// TIA Portal V17 export
// export: Created 2025-03-10T12:18:24.9535998Z, ExportSetting WithDefaults, DisplayName Totally Integrated Automation Portal, DisplayVersion V17 Update 8, DisplayName TIA Portal Openness, DisplayVersion V17 Update 8, DisplayName TIA Portal Version Control Interface, DisplayVersion V17, DisplayName SINAMICS Startdrive Advanced, DisplayVersion V17 SP2, DisplayName SINAMICS Startdrive G110M, G120, G120C, G120D, G120P, G115D, DisplayVersion V17 SP2, DisplayName SINAMICS Startdrive G130, G150, S120, S150, SINAMICS MV, S210, DisplayVersion V17 SP2, DisplayName STEP 7 Professional, DisplayVersion V17 Update 8, DisplayName SINUMERIK ONE STEP 7 Toolbox, DisplayVersion V17 Update 12, DisplayName SINUMERIK 840D sl STEP 7 Toolbox, DisplayVersion V17 Update 12, DisplayName STEP 7 Safety, DisplayVersion V17 Update 6, DisplayName WinCC Advanced, DisplayVersion V17 Update 8
DATA_BLOCK "DB428_OPERATOR_HELP"   // DB428
{ S7_Optimized_Access := 'FALSE' }
VERSION : 1.0
// stored: AutoNumber false, DBAccessibleFromOPCUA true, DBAccessibleFromWebserver true, IsOnlyStoredInLoadMemory false, IsWriteProtectedInAS false
   VAR RETAIN
      HELP_OPERATOR_0 : Bool;   // EMPTY
      HELP_OPERATOR_1 : Bool;   // EMPTY
      HELP_OPERATOR_2 : Bool;
      HELP_OPERATOR_3 : Bool;
      HELP_OPERATOR_4 : Bool;
      HELP_OPERATOR_5 : Bool;
      HELP_OPERATOR_6 : Bool;
      HELP_OPERATOR_7 : Bool;
      HELP_OPERATOR_8 : Bool;
      HELP_OPERATOR_9 : Bool;
      HELP_OPERATOR_10 : Bool;
      HELP_OPERATOR_11 : Bool;
      HELP_OPERATOR_12 : Bool;
      HELP_OPERATOR_13 : Bool;
      HELP_OPERATOR_14 : Bool;
      HELP_OPERATOR_15 : Bool;
      HELP_OPERATOR_16 : Bool;
      HELP_OPERATOR_17 : Bool;
      HELP_OPERATOR_18 : Bool;
      HELP_OPERATOR_19 : Bool;
      HELP_OPERATOR_20 : Bool;
      HELP_OPERATOR_21 : Bool;
      HELP_OPERATOR_22 : Bool;
      HELP_OPERATOR_23 : Bool;
      HELP_OPERATOR_24 : Bool;
      HELP_OPERATOR_25 : Bool;
      HELP_OPERATOR_26 : Bool;
      HELP_OPERATOR_27 : Bool;
      HELP_OPERATOR_28 : Bool;
      HELP_OPERATOR_29 : Bool;
      HELP_OPERATOR_30 : Bool;
      HELP_OPERATOR_31 : Bool;
      HELP_OPERATOR_32 : Bool;
      HELP_OPERATOR_33 : Bool;
      HELP_OPERATOR_34 : Bool;
      HELP_OPERATOR_35 : Bool;
      HELP_OPERATOR_36 : Bool;
      HELP_OPERATOR_37 : Bool;
      HELP_OPERATOR_38 : Bool;
      HELP_OPERATOR_39 : Bool;
      HELP_OPERATOR_40 : Bool;
      HELP_OPERATOR_41 : Bool;
      HELP_OPERATOR_42 : Bool;
      HELP_OPERATOR_43 : Bool;
      HELP_OPERATOR_44 : Bool;
      HELP_OPERATOR_45 : Bool;
      HELP_OPERATOR_46 : Bool;
      HELP_OPERATOR_47 : Bool;
      HELP_OPERATOR_48 : Bool;
      HELP_OPERATOR_49 : Bool;
      HELP_OPERATOR_50 : Bool;
      HELP_OPERATOR_51 : Bool;
      HELP_OPERATOR_52 : Bool;
      HELP_OPERATOR_53 : Bool;
      HELP_OPERATOR_54 : Bool;
      HELP_OPERATOR_55 : Bool;
      HELP_OPERATOR_56 : Bool;
      HELP_OPERATOR_57 : Bool;
      HELP_OPERATOR_58 : Bool;
      HELP_OPERATOR_59 : Bool;
      HELP_OPERATOR_60 : Bool;
      HELP_OPERATOR_61 : Bool;
      HELP_OPERATOR_62 : Bool;
      HELP_OPERATOR_63 : Bool;
      HELP_OPERATOR_64 : Bool;
      HELP_OPERATOR_65 : Bool;
      HELP_OPERATOR_66 : Bool;
      HELP_OPERATOR_67 : Bool;
      HELP_OPERATOR_68 : Bool;
      HELP_OPERATOR_69 : Bool;
      HELP_OPERATOR_70 : Bool;
      HELP_OPERATOR_71 : Bool;
      HELP_OPERATOR_72 : Bool;
      HELP_OPERATOR_73 : Bool;
      HELP_OPERATOR_74 : Bool;
      HELP_OPERATOR_75 : Bool;
      HELP_OPERATOR_76 : Bool;
      HELP_OPERATOR_77 : Bool;
      HELP_OPERATOR_78 : Bool;
      HELP_OPERATOR_79 : Bool;
      HELP_OPERATOR_80 : Bool;
      HELP_OPERATOR_81 : Bool;
      HELP_OPERATOR_82 : Bool;
      HELP_OPERATOR_83 : Bool;
      HELP_OPERATOR_84 : Bool;
      HELP_OPERATOR_85 : Bool;
      HELP_OPERATOR_86 : Bool;
      HELP_OPERATOR_87 : Bool;
      HELP_OPERATOR_88 : Bool;
      HELP_OPERATOR_89 : Bool;
      HELP_OPERATOR_90 : Bool;
      HELP_OPERATOR_91 : Bool;
      HELP_OPERATOR_92 : Bool;
      HELP_OPERATOR_93 : Bool;
      HELP_OPERATOR_94 : Bool;
      HELP_OPERATOR_95 : Bool;
      HELP_OPERATOR_96 : Bool;
      HELP_OPERATOR_97 : Bool;
      HELP_OPERATOR_98 : Bool;
      HELP_OPERATOR_99 : Bool;
      HELP_OPERATOR_100 : Bool;
      HELP_OPERATOR_101 : Bool;
      HELP_OPERATOR_102 : Bool;
      HELP_OPERATOR_103 : Bool;
      HELP_OPERATOR_104 : Bool;
      HELP_OPERATOR_105 : Bool;
      HELP_OPERATOR_106 : Bool;
      HELP_OPERATOR_107 : Bool;
      HELP_OPERATOR_108 : Bool;
      HELP_OPERATOR_109 : Bool;
      HELP_OPERATOR_110 : Bool;
      HELP_OPERATOR_111 : Bool;
      HELP_OPERATOR_112 : Bool;
      HELP_OPERATOR_113 : Bool;
      HELP_OPERATOR_114 : Bool;
      HELP_OPERATOR_115 : Bool;
      HELP_OPERATOR_116 : Bool;
      HELP_OPERATOR_117 : Bool;
      HELP_OPERATOR_118 : Bool;
      HELP_OPERATOR_119 : Bool;
      HELP_OPERATOR_120 : Bool;
      HELP_OPERATOR_121 : Bool;
      HELP_OPERATOR_122 : Bool;
      HELP_OPERATOR_123 : Bool;
      HELP_OPERATOR_124 : Bool;
      HELP_OPERATOR_125 : Bool;
      HELP_OPERATOR_126 : Bool;
      HELP_OPERATOR_127 : Bool;
      HELP_OPERATOR_128 : Bool;
      HELP_OPERATOR_129 : Bool;
      HELP_OPERATOR_130 : Bool;
      HELP_OPERATOR_131 : Bool;
      HELP_OPERATOR_132 : Bool;
      HELP_OPERATOR_133 : Bool;
      HELP_OPERATOR_134 : Bool;
      HELP_OPERATOR_135 : Bool;
      HELP_OPERATOR_136 : Bool;
      HELP_OPERATOR_137 : Bool;
      HELP_OPERATOR_138 : Bool;
      HELP_OPERATOR_139 : Bool;
      HELP_OPERATOR_140 : Bool;
      HELP_OPERATOR_141 : Bool;
      HELP_OPERATOR_142 : Bool;
      HELP_OPERATOR_143 : Bool;
      HELP_OPERATOR_144 : Bool;
      HELP_OPERATOR_145 : Bool;
      HELP_OPERATOR_146 : Bool;
      HELP_OPERATOR_147 : Bool;
      HELP_OPERATOR_148 : Bool;
      HELP_OPERATOR_149 : Bool;
      HELP_OPERATOR_150 : Bool;   // RETURN UNIT 1 TO HOME POSITION
      HELP_OPERATOR_151 : Bool;   // RETURN UNIT 2 TO HOME POSITION
      HELP_OPERATOR_152 : Bool;   // RETURN UNIT 3 TO HOME POSITION
      HELP_OPERATOR_153 : Bool;   // RETURN UNIT 4 TO HOME POSITION
      HELP_OPERATOR_154 : Bool;   // RETURN UNIT 5 TO HOME POSITION
      HELP_OPERATOR_155 : Bool;   // RETURN UNIT 6 TO HOME POSITION
      HELP_OPERATOR_156 : Bool;   // RETURN UNIT 7 TO HOME POSITION
      HELP_OPERATOR_157 : Bool;   // RETURN UNIT 8 TO HOME POSITION
      HELP_OPERATOR_158 : Bool;   // RETURN UNIT 9 TO HOME POSITION
      HELP_OPERATOR_159 : Bool;   // RETURN UNIT 10 TO HOME POSITION
      HELP_OPERATOR_160 : Bool;
      HELP_OPERATOR_161 : Bool;
      HELP_OPERATOR_162 : Bool;   // UNIT 1 IN HOME POSITION
      HELP_OPERATOR_163 : Bool;   // UNIT 2 IN HOME POSITION
      HELP_OPERATOR_164 : Bool;   // UNIT 3 IN HOME POSITION
      HELP_OPERATOR_165 : Bool;   // UNIT 4 IN HOME POSITION
      HELP_OPERATOR_166 : Bool;   // UNIT 5 IN HOME POSITION
      HELP_OPERATOR_167 : Bool;   // UNIT 6 IN HOME POSITION
      HELP_OPERATOR_168 : Bool;   // UNIT 7 IN HOME POSITION
      HELP_OPERATOR_169 : Bool;   // UNIT 8 IN HOME POSITION
      HELP_OPERATOR_170 : Bool;   // UNIT 9 IN HOME POSITION
      HELP_OPERATOR_171 : Bool;   // UNIT 10 IN HOME POSITION
      HELP_OPERATOR_172 : Bool;
      HELP_OPERATOR_173 : Bool;
      HELP_OPERATOR_174 : Bool;   // UNIT 01R SPINDLES NOT STOPPED
      HELP_OPERATOR_175 : Bool;   // UNIT 01L SPINDLES NOT STOPPED
      HELP_OPERATOR_176 : Bool;
      HELP_OPERATOR_177 : Bool;
      HELP_OPERATOR_178 : Bool;   // TOOLS IN MAGAZINE 01R NOT OK
      HELP_OPERATOR_179 : Bool;   // TOOLS IN MAGAZINE 01L NOT OK
      HELP_OPERATOR_180 : Bool;
      HELP_OPERATOR_181 : Bool;
      HELP_OPERATOR_182 : Bool;   // RETURN MACHINE TO HOME POSITION
      HELP_OPERATOR_183 : Bool;
      HELP_OPERATOR_184 : Bool;   // RETURN PART HANDLING DEVICE TO HOME POSITION
      HELP_OPERATOR_185 : Bool;   // PART HANDLING DEVICE IN HOME POSITION
      HELP_OPERATOR_186 : Bool;   // ADVANCE PHD TO LOAD UNLOAD POS FIXTURE
      HELP_OPERATOR_187 : Bool;
      HELP_OPERATOR_188 : Bool;
      HELP_OPERATOR_189 : Bool;
      HELP_OPERATOR_190 : Bool;   // NO PART AT FEED
      HELP_OPERATOR_191 : Bool;   // PARTS DELIVERY OCCUPIED
      HELP_OPERATOR_192 : Bool;
      HELP_OPERATOR_193 : Bool;
      HELP_OPERATOR_194 : Bool;
      HELP_OPERATOR_195 : Bool;
      HELP_OPERATOR_196 : Bool;
      HELP_OPERATOR_197 : Bool;
      HELP_OPERATOR_198 : Bool;
      HELP_OPERATOR_199 : Bool;
      HELP_OPERATOR_200 : Bool;   // SELECT MANUAL MODE
      HELP_OPERATOR_201 : Bool;   // SELECT JOG MODE
      HELP_OPERATOR_202 : Bool;   // SELECT SEMIAUTOMATIC MODE
      HELP_OPERATOR_203 : Bool;   // SELECT TOOL CHANGE MODE
      HELP_OPERATOR_204 : Bool;   // SELECT AUTOMATIC MODE
      HELP_OPERATOR_205 : Bool;   // SELECT INCREMENTAL MODE
      HELP_OPERATOR_206 : Bool;   // SELECT AUTO. OR SEMIAUTO. OR SINGLE MODE
      HELP_OPERATOR_207 : Bool;
      HELP_OPERATOR_208 : Bool;
      HELP_OPERATOR_209 : Bool;
      HELP_OPERATOR_210 : Bool;
      HELP_OPERATOR_211 : Bool;
      HELP_OPERATOR_212 : Bool;
      HELP_OPERATOR_213 : Bool;
      HELP_OPERATOR_214 : Bool;
      HELP_OPERATOR_215 : Bool;   // UNSELECT REFERENCE MODE
      HELP_OPERATOR_216 : Bool;   // UNSELECT STEP BY STEP MODE
      HELP_OPERATOR_217 : Bool;   // UNSELECT MANUAL LOADING CYCLE
      HELP_OPERATOR_218 : Bool;   // UNSELECT MDA MODE
      HELP_OPERATOR_219 : Bool;   // UNSELECT RUN-OUT CYCLE
      HELP_OPERATOR_220 : Bool;   // UNSELECT DRY CYCLE
      HELP_OPERATOR_221 : Bool;   // UNSELECT GANTRY TEST CYCLE
      HELP_OPERATOR_222 : Bool;   // UNSELECT ROBOT DRY CYCLE
      HELP_OPERATOR_223 : Bool;   // UNSELECT SINGLE CYCLE
      HELP_OPERATOR_224 : Bool;
      HELP_OPERATOR_225 : Bool;
      HELP_OPERATOR_226 : Bool;
      HELP_OPERATOR_227 : Bool;
      HELP_OPERATOR_228 : Bool;
      HELP_OPERATOR_229 : Bool;
      HELP_OPERATOR_230 : Bool;   // ENABLE BA1 MODE
      HELP_OPERATOR_231 : Bool;   // ENABLE BA1 OR BA3 MODE
      HELP_OPERATOR_232 : Bool;   // ENABLE BA2 MODE OR CLOSE SAFETY DOORS
      HELP_OPERATOR_233 : Bool;
      HELP_OPERATOR_234 : Bool;
      HELP_OPERATOR_235 : Bool;
      HELP_OPERATOR_236 : Bool;
      HELP_OPERATOR_237 : Bool;
      HELP_OPERATOR_238 : Bool;
      HELP_OPERATOR_239 : Bool;
      HELP_OPERATOR_240 : Bool;
      HELP_OPERATOR_241 : Bool;
      HELP_OPERATOR_242 : Bool;
      HELP_OPERATOR_243 : Bool;
      HELP_OPERATOR_244 : Bool;
      HELP_OPERATOR_245 : Bool;
      HELP_OPERATOR_246 : Bool;
      HELP_OPERATOR_247 : Bool;
      HELP_OPERATOR_248 : Bool;
      HELP_OPERATOR_249 : Bool;
      HELP_OPERATOR_250 : Bool;   // MAIN OPERATOR PANEL, PRESS BUTTON CONTROL ON
      HELP_OPERATOR_251 : Bool;   // MAIN OPERATOR PANEL, PRESS BUTTON RESET
      HELP_OPERATOR_252 : Bool;   // REMOVE EMERGENCY STOPS, PRESS RESET FAULTS
      HELP_OPERATOR_253 : Bool;   // MACHINE STOP SERVICES DELAYED ENABLED
      HELP_OPERATOR_254 : Bool;   // SWITCH ON PNEUMATIC SYSTEM
      HELP_OPERATOR_255 : Bool;
      HELP_OPERATOR_256 : Bool;
      HELP_OPERATOR_257 : Bool;
      HELP_OPERATOR_258 : Bool;
      HELP_OPERATOR_259 : Bool;
      HELP_OPERATOR_260 : Bool;
      HELP_OPERATOR_261 : Bool;
      HELP_OPERATOR_262 : Bool;
      HELP_OPERATOR_263 : Bool;
      HELP_OPERATOR_264 : Bool;
      HELP_OPERATOR_265 : Bool;
      HELP_OPERATOR_266 : Bool;
      HELP_OPERATOR_267 : Bool;
      HELP_OPERATOR_268 : Bool;
      HELP_OPERATOR_269 : Bool;
      HELP_OPERATOR_270 : Bool;
      HELP_OPERATOR_271 : Bool;
      HELP_OPERATOR_272 : Bool;
      HELP_OPERATOR_273 : Bool;
      HELP_OPERATOR_274 : Bool;
      HELP_OPERATOR_275 : Bool;
      HELP_OPERATOR_276 : Bool;
      HELP_OPERATOR_277 : Bool;
      HELP_OPERATOR_278 : Bool;
      HELP_OPERATOR_279 : Bool;
      HELP_OPERATOR_280 : Bool;
      HELP_OPERATOR_281 : Bool;
      HELP_OPERATOR_282 : Bool;
      HELP_OPERATOR_283 : Bool;
      HELP_OPERATOR_284 : Bool;
      HELP_OPERATOR_285 : Bool;
      HELP_OPERATOR_286 : Bool;
      HELP_OPERATOR_287 : Bool;
      HELP_OPERATOR_288 : Bool;
      HELP_OPERATOR_289 : Bool;
      HELP_OPERATOR_290 : Bool;
      HELP_OPERATOR_291 : Bool;
      HELP_OPERATOR_292 : Bool;
      HELP_OPERATOR_293 : Bool;
      HELP_OPERATOR_294 : Bool;
      HELP_OPERATOR_295 : Bool;
      HELP_OPERATOR_296 : Bool;
      HELP_OPERATOR_297 : Bool;
      HELP_OPERATOR_298 : Bool;
      HELP_OPERATOR_299 : Bool;
      HELP_OPERATOR_300 : Bool;
      HELP_OPERATOR_301 : Bool;
      HELP_OPERATOR_302 : Bool;
      HELP_OPERATOR_303 : Bool;
      HELP_OPERATOR_304 : Bool;
      HELP_OPERATOR_305 : Bool;
      HELP_OPERATOR_306 : Bool;
      HELP_OPERATOR_307 : Bool;
      HELP_OPERATOR_308 : Bool;
      HELP_OPERATOR_309 : Bool;
      HELP_OPERATOR_310 : Bool;
      HELP_OPERATOR_311 : Bool;
      HELP_OPERATOR_312 : Bool;
      HELP_OPERATOR_313 : Bool;
      HELP_OPERATOR_314 : Bool;
      HELP_OPERATOR_315 : Bool;
      HELP_OPERATOR_316 : Bool;
      HELP_OPERATOR_317 : Bool;
      HELP_OPERATOR_318 : Bool;
      HELP_OPERATOR_319 : Bool;
      HELP_OPERATOR_320 : Bool;
      HELP_OPERATOR_321 : Bool;
      HELP_OPERATOR_322 : Bool;
      HELP_OPERATOR_323 : Bool;
      HELP_OPERATOR_324 : Bool;
      HELP_OPERATOR_325 : Bool;
      HELP_OPERATOR_326 : Bool;
      HELP_OPERATOR_327 : Bool;
      HELP_OPERATOR_328 : Bool;
      HELP_OPERATOR_329 : Bool;
      HELP_OPERATOR_330 : Bool;
      HELP_OPERATOR_331 : Bool;
      HELP_OPERATOR_332 : Bool;
      HELP_OPERATOR_333 : Bool;
      HELP_OPERATOR_334 : Bool;
      HELP_OPERATOR_335 : Bool;
      HELP_OPERATOR_336 : Bool;
      HELP_OPERATOR_337 : Bool;
      HELP_OPERATOR_338 : Bool;
      HELP_OPERATOR_339 : Bool;
      HELP_OPERATOR_340 : Bool;
      HELP_OPERATOR_341 : Bool;
      HELP_OPERATOR_342 : Bool;
      HELP_OPERATOR_343 : Bool;
      HELP_OPERATOR_344 : Bool;
      HELP_OPERATOR_345 : Bool;
      HELP_OPERATOR_346 : Bool;
      HELP_OPERATOR_347 : Bool;
      HELP_OPERATOR_348 : Bool;
      HELP_OPERATOR_349 : Bool;
      HELP_OPERATOR_350 : Bool;
      HELP_OPERATOR_351 : Bool;
      HELP_OPERATOR_352 : Bool;
      HELP_OPERATOR_353 : Bool;
      HELP_OPERATOR_354 : Bool;
      HELP_OPERATOR_355 : Bool;
      HELP_OPERATOR_356 : Bool;
      HELP_OPERATOR_357 : Bool;
      HELP_OPERATOR_358 : Bool;
      HELP_OPERATOR_359 : Bool;
      HELP_OPERATOR_360 : Bool;
      HELP_OPERATOR_361 : Bool;
      HELP_OPERATOR_362 : Bool;
      HELP_OPERATOR_363 : Bool;
      HELP_OPERATOR_364 : Bool;
      HELP_OPERATOR_365 : Bool;
      HELP_OPERATOR_366 : Bool;
      HELP_OPERATOR_367 : Bool;
      HELP_OPERATOR_368 : Bool;
      HELP_OPERATOR_369 : Bool;
      HELP_OPERATOR_370 : Bool;
      HELP_OPERATOR_371 : Bool;
      HELP_OPERATOR_372 : Bool;
      HELP_OPERATOR_373 : Bool;
      HELP_OPERATOR_374 : Bool;
      HELP_OPERATOR_375 : Bool;
      HELP_OPERATOR_376 : Bool;
      HELP_OPERATOR_377 : Bool;
      HELP_OPERATOR_378 : Bool;
      HELP_OPERATOR_379 : Bool;
      HELP_OPERATOR_380 : Bool;
      HELP_OPERATOR_381 : Bool;
      HELP_OPERATOR_382 : Bool;
      HELP_OPERATOR_383 : Bool;
      HELP_OPERATOR_384 : Bool;
      HELP_OPERATOR_385 : Bool;
      HELP_OPERATOR_386 : Bool;
      HELP_OPERATOR_387 : Bool;
      HELP_OPERATOR_388 : Bool;
      HELP_OPERATOR_389 : Bool;
      HELP_OPERATOR_390 : Bool;
      HELP_OPERATOR_391 : Bool;
      HELP_OPERATOR_392 : Bool;
      HELP_OPERATOR_393 : Bool;
      HELP_OPERATOR_394 : Bool;
      HELP_OPERATOR_395 : Bool;
      HELP_OPERATOR_396 : Bool;
      HELP_OPERATOR_397 : Bool;
      HELP_OPERATOR_398 : Bool;
      HELP_OPERATOR_399 : Bool;
      HELP_OPERATOR_400 : Bool;
      HELP_OPERATOR_401 : Bool;
      HELP_OPERATOR_402 : Bool;
      HELP_OPERATOR_403 : Bool;
      HELP_OPERATOR_404 : Bool;
      HELP_OPERATOR_405 : Bool;
      HELP_OPERATOR_406 : Bool;
      HELP_OPERATOR_407 : Bool;
      HELP_OPERATOR_408 : Bool;
      HELP_OPERATOR_409 : Bool;
      HELP_OPERATOR_410 : Bool;
      HELP_OPERATOR_411 : Bool;
      HELP_OPERATOR_412 : Bool;
      HELP_OPERATOR_413 : Bool;
      HELP_OPERATOR_414 : Bool;
      HELP_OPERATOR_415 : Bool;
      HELP_OPERATOR_416 : Bool;
      HELP_OPERATOR_417 : Bool;
      HELP_OPERATOR_418 : Bool;
      HELP_OPERATOR_419 : Bool;
      HELP_OPERATOR_420 : Bool;
      HELP_OPERATOR_421 : Bool;
      HELP_OPERATOR_422 : Bool;
      HELP_OPERATOR_423 : Bool;
      HELP_OPERATOR_424 : Bool;
      HELP_OPERATOR_425 : Bool;
      HELP_OPERATOR_426 : Bool;
      HELP_OPERATOR_427 : Bool;
      HELP_OPERATOR_428 : Bool;
      HELP_OPERATOR_429 : Bool;
      HELP_OPERATOR_430 : Bool;
      HELP_OPERATOR_431 : Bool;
      HELP_OPERATOR_432 : Bool;
      HELP_OPERATOR_433 : Bool;
      HELP_OPERATOR_434 : Bool;
      HELP_OPERATOR_435 : Bool;
      HELP_OPERATOR_436 : Bool;
      HELP_OPERATOR_437 : Bool;
      HELP_OPERATOR_438 : Bool;
      HELP_OPERATOR_439 : Bool;
      HELP_OPERATOR_440 : Bool;
      HELP_OPERATOR_441 : Bool;
      HELP_OPERATOR_442 : Bool;
      HELP_OPERATOR_443 : Bool;
      HELP_OPERATOR_444 : Bool;
      HELP_OPERATOR_445 : Bool;
      HELP_OPERATOR_446 : Bool;
      HELP_OPERATOR_447 : Bool;
      HELP_OPERATOR_448 : Bool;
      HELP_OPERATOR_449 : Bool;
      HELP_OPERATOR_450 : Bool;
      HELP_OPERATOR_451 : Bool;
      HELP_OPERATOR_452 : Bool;
      HELP_OPERATOR_453 : Bool;
      HELP_OPERATOR_454 : Bool;
      HELP_OPERATOR_455 : Bool;
      HELP_OPERATOR_456 : Bool;
      HELP_OPERATOR_457 : Bool;
      HELP_OPERATOR_458 : Bool;
      HELP_OPERATOR_459 : Bool;
      HELP_OPERATOR_460 : Bool;
      HELP_OPERATOR_461 : Bool;
      HELP_OPERATOR_462 : Bool;
      HELP_OPERATOR_463 : Bool;
      HELP_OPERATOR_464 : Bool;
      HELP_OPERATOR_465 : Bool;
      HELP_OPERATOR_466 : Bool;
      HELP_OPERATOR_467 : Bool;
      HELP_OPERATOR_468 : Bool;
      HELP_OPERATOR_469 : Bool;
      HELP_OPERATOR_470 : Bool;
      HELP_OPERATOR_471 : Bool;
      HELP_OPERATOR_472 : Bool;
      HELP_OPERATOR_473 : Bool;
      HELP_OPERATOR_474 : Bool;
      HELP_OPERATOR_475 : Bool;
      HELP_OPERATOR_476 : Bool;
      HELP_OPERATOR_477 : Bool;
      HELP_OPERATOR_478 : Bool;
      HELP_OPERATOR_479 : Bool;
      HELP_OPERATOR_480 : Bool;
      HELP_OPERATOR_481 : Bool;
      HELP_OPERATOR_482 : Bool;
      HELP_OPERATOR_483 : Bool;
      HELP_OPERATOR_484 : Bool;
      HELP_OPERATOR_485 : Bool;
      HELP_OPERATOR_486 : Bool;
      HELP_OPERATOR_487 : Bool;
      HELP_OPERATOR_488 : Bool;
      HELP_OPERATOR_489 : Bool;
      HELP_OPERATOR_490 : Bool;
      HELP_OPERATOR_491 : Bool;
      HELP_OPERATOR_492 : Bool;
      HELP_OPERATOR_493 : Bool;
      HELP_OPERATOR_494 : Bool;
      HELP_OPERATOR_495 : Bool;
      HELP_OPERATOR_496 : Bool;
      HELP_OPERATOR_497 : Bool;
      HELP_OPERATOR_498 : Bool;
      HELP_OPERATOR_499 : Bool;
      HELP_OPERATOR_500 : Bool;
      HELP_OPERATOR_501 : Bool;
      HELP_OPERATOR_502 : Bool;
      HELP_OPERATOR_503 : Bool;
      HELP_OPERATOR_504 : Bool;
      HELP_OPERATOR_505 : Bool;
      HELP_OPERATOR_506 : Bool;
      HELP_OPERATOR_507 : Bool;
      HELP_OPERATOR_508 : Bool;
      HELP_OPERATOR_509 : Bool;
      HELP_OPERATOR_510 : Bool;
      HELP_OPERATOR_511 : Bool;
      HELP_OPERATOR_512 : Bool;
      HELP_OPERATOR_513 : Bool;
      HELP_OPERATOR_514 : Bool;
      HELP_OPERATOR_515 : Bool;
      HELP_OPERATOR_516 : Bool;
      HELP_OPERATOR_517 : Bool;
      HELP_OPERATOR_518 : Bool;
      HELP_OPERATOR_519 : Bool;
      HELP_OPERATOR_520 : Bool;
      HELP_OPERATOR_521 : Bool;
      HELP_OPERATOR_522 : Bool;
      HELP_OPERATOR_523 : Bool;
      HELP_OPERATOR_524 : Bool;
      HELP_OPERATOR_525 : Bool;
      HELP_OPERATOR_526 : Bool;
      HELP_OPERATOR_527 : Bool;
      HELP_OPERATOR_528 : Bool;
      HELP_OPERATOR_529 : Bool;
      HELP_OPERATOR_530 : Bool;
      HELP_OPERATOR_531 : Bool;   // STIRRER MOTOR NOT ENABLED
      HELP_OPERATOR_532 : Bool;   // STIRRER FAULT
      HELP_OPERATOR_533 : Bool;   // STIRRER ON
      HELP_OPERATOR_534 : Bool;   // STIRRER STOP GENERAL CONDITIONS MISSING
      HELP_OPERATOR_535 : Bool;   // STIRRER OFF
      HELP_OPERATOR_536 : Bool;
      HELP_OPERATOR_537 : Bool;
      HELP_OPERATOR_538 : Bool;
      HELP_OPERATOR_539 : Bool;
      HELP_OPERATOR_540 : Bool;   // TEMPERATURE JACKET BREAKER TRIPPED
      HELP_OPERATOR_541 : Bool;
      HELP_OPERATOR_542 : Bool;
      HELP_OPERATOR_543 : Bool;
      HELP_OPERATOR_544 : Bool;
      HELP_OPERATOR_545 : Bool;
      HELP_OPERATOR_546 : Bool;
      HELP_OPERATOR_547 : Bool;
      HELP_OPERATOR_548 : Bool;
      HELP_OPERATOR_549 : Bool;
      HELP_OPERATOR_550 : Bool;
      HELP_OPERATOR_551 : Bool;
      HELP_OPERATOR_552 : Bool;
      HELP_OPERATOR_553 : Bool;
      HELP_OPERATOR_554 : Bool;
      HELP_OPERATOR_555 : Bool;
      HELP_OPERATOR_556 : Bool;
      HELP_OPERATOR_557 : Bool;
      HELP_OPERATOR_558 : Bool;
      HELP_OPERATOR_559 : Bool;
      HELP_OPERATOR_560 : Bool;
      HELP_OPERATOR_561 : Bool;
      HELP_OPERATOR_562 : Bool;
      HELP_OPERATOR_563 : Bool;
      HELP_OPERATOR_564 : Bool;
      HELP_OPERATOR_565 : Bool;
      HELP_OPERATOR_566 : Bool;
      HELP_OPERATOR_567 : Bool;
      HELP_OPERATOR_568 : Bool;
      HELP_OPERATOR_569 : Bool;
      HELP_OPERATOR_570 : Bool;
      HELP_OPERATOR_571 : Bool;
      HELP_OPERATOR_572 : Bool;
      HELP_OPERATOR_573 : Bool;
      HELP_OPERATOR_574 : Bool;
      HELP_OPERATOR_575 : Bool;
      HELP_OPERATOR_576 : Bool;
      HELP_OPERATOR_577 : Bool;
      HELP_OPERATOR_578 : Bool;
      HELP_OPERATOR_579 : Bool;
      HELP_OPERATOR_580 : Bool;
      HELP_OPERATOR_581 : Bool;
      HELP_OPERATOR_582 : Bool;
      HELP_OPERATOR_583 : Bool;
      HELP_OPERATOR_584 : Bool;
      HELP_OPERATOR_585 : Bool;
      HELP_OPERATOR_586 : Bool;
      HELP_OPERATOR_587 : Bool;
      HELP_OPERATOR_588 : Bool;
      HELP_OPERATOR_589 : Bool;
      HELP_OPERATOR_590 : Bool;
      HELP_OPERATOR_591 : Bool;
      HELP_OPERATOR_592 : Bool;
      HELP_OPERATOR_593 : Bool;
      HELP_OPERATOR_594 : Bool;
      HELP_OPERATOR_595 : Bool;
      HELP_OPERATOR_596 : Bool;
      HELP_OPERATOR_597 : Bool;
      HELP_OPERATOR_598 : Bool;
      HELP_OPERATOR_599 : Bool;
      HELP_OPERATOR_600 : Bool;
      HELP_OPERATOR_601 : Bool;
      HELP_OPERATOR_602 : Bool;
      HELP_OPERATOR_603 : Bool;
      HELP_OPERATOR_604 : Bool;
      HELP_OPERATOR_605 : Bool;
      HELP_OPERATOR_606 : Bool;
      HELP_OPERATOR_607 : Bool;
      HELP_OPERATOR_608 : Bool;
      HELP_OPERATOR_609 : Bool;
      HELP_OPERATOR_610 : Bool;
      HELP_OPERATOR_611 : Bool;
      HELP_OPERATOR_612 : Bool;
      HELP_OPERATOR_613 : Bool;
      HELP_OPERATOR_614 : Bool;
      HELP_OPERATOR_615 : Bool;
      HELP_OPERATOR_616 : Bool;
      HELP_OPERATOR_617 : Bool;
      HELP_OPERATOR_618 : Bool;
      HELP_OPERATOR_619 : Bool;
      HELP_OPERATOR_620 : Bool;
      HELP_OPERATOR_621 : Bool;
      HELP_OPERATOR_622 : Bool;
      HELP_OPERATOR_623 : Bool;
      HELP_OPERATOR_624 : Bool;
      HELP_OPERATOR_625 : Bool;
      HELP_OPERATOR_626 : Bool;
      HELP_OPERATOR_627 : Bool;
      HELP_OPERATOR_628 : Bool;
      HELP_OPERATOR_629 : Bool;
      HELP_OPERATOR_630 : Bool;
      HELP_OPERATOR_631 : Bool;
      HELP_OPERATOR_632 : Bool;
      HELP_OPERATOR_633 : Bool;
      HELP_OPERATOR_634 : Bool;
      HELP_OPERATOR_635 : Bool;
      HELP_OPERATOR_636 : Bool;
      HELP_OPERATOR_637 : Bool;
      HELP_OPERATOR_638 : Bool;
      HELP_OPERATOR_639 : Bool;
      HELP_OPERATOR_640 : Bool;
      HELP_OPERATOR_641 : Bool;
      HELP_OPERATOR_642 : Bool;
      HELP_OPERATOR_643 : Bool;
      HELP_OPERATOR_644 : Bool;
      HELP_OPERATOR_645 : Bool;
      HELP_OPERATOR_646 : Bool;
      HELP_OPERATOR_647 : Bool;
      HELP_OPERATOR_648 : Bool;
      HELP_OPERATOR_649 : Bool;
      HELP_OPERATOR_650 : Bool;
      HELP_OPERATOR_651 : Bool;
      HELP_OPERATOR_652 : Bool;
      HELP_OPERATOR_653 : Bool;
      HELP_OPERATOR_654 : Bool;
      HELP_OPERATOR_655 : Bool;
      HELP_OPERATOR_656 : Bool;
      HELP_OPERATOR_657 : Bool;
      HELP_OPERATOR_658 : Bool;
      HELP_OPERATOR_659 : Bool;
      HELP_OPERATOR_660 : Bool;
      HELP_OPERATOR_661 : Bool;
      HELP_OPERATOR_662 : Bool;
      HELP_OPERATOR_663 : Bool;
      HELP_OPERATOR_664 : Bool;
      HELP_OPERATOR_665 : Bool;
      HELP_OPERATOR_666 : Bool;
      HELP_OPERATOR_667 : Bool;
      HELP_OPERATOR_668 : Bool;
      HELP_OPERATOR_669 : Bool;
      HELP_OPERATOR_670 : Bool;
      HELP_OPERATOR_671 : Bool;
      HELP_OPERATOR_672 : Bool;
      HELP_OPERATOR_673 : Bool;
      HELP_OPERATOR_674 : Bool;
      HELP_OPERATOR_675 : Bool;
      HELP_OPERATOR_676 : Bool;
      HELP_OPERATOR_677 : Bool;
      HELP_OPERATOR_678 : Bool;
      HELP_OPERATOR_679 : Bool;
      HELP_OPERATOR_680 : Bool;
      HELP_OPERATOR_681 : Bool;
      HELP_OPERATOR_682 : Bool;
      HELP_OPERATOR_683 : Bool;
      HELP_OPERATOR_684 : Bool;
      HELP_OPERATOR_685 : Bool;
      HELP_OPERATOR_686 : Bool;
      HELP_OPERATOR_687 : Bool;
      HELP_OPERATOR_688 : Bool;
      HELP_OPERATOR_689 : Bool;
      HELP_OPERATOR_690 : Bool;
      HELP_OPERATOR_691 : Bool;
      HELP_OPERATOR_692 : Bool;
      HELP_OPERATOR_693 : Bool;
      HELP_OPERATOR_694 : Bool;
      HELP_OPERATOR_695 : Bool;
      HELP_OPERATOR_696 : Bool;
      HELP_OPERATOR_697 : Bool;
      HELP_OPERATOR_698 : Bool;
      HELP_OPERATOR_699 : Bool;
      HELP_OPERATOR_700 : Bool;
      HELP_OPERATOR_701 : Bool;
      HELP_OPERATOR_702 : Bool;
      HELP_OPERATOR_703 : Bool;
      HELP_OPERATOR_704 : Bool;
      HELP_OPERATOR_705 : Bool;
      HELP_OPERATOR_706 : Bool;
      HELP_OPERATOR_707 : Bool;
      HELP_OPERATOR_708 : Bool;
      HELP_OPERATOR_709 : Bool;
      HELP_OPERATOR_710 : Bool;
      HELP_OPERATOR_711 : Bool;
      HELP_OPERATOR_712 : Bool;
      HELP_OPERATOR_713 : Bool;
      HELP_OPERATOR_714 : Bool;
      HELP_OPERATOR_715 : Bool;
      HELP_OPERATOR_716 : Bool;
      HELP_OPERATOR_717 : Bool;
      HELP_OPERATOR_718 : Bool;
      HELP_OPERATOR_719 : Bool;
      HELP_OPERATOR_720 : Bool;
      HELP_OPERATOR_721 : Bool;
      HELP_OPERATOR_722 : Bool;
      HELP_OPERATOR_723 : Bool;
      HELP_OPERATOR_724 : Bool;
      HELP_OPERATOR_725 : Bool;
      HELP_OPERATOR_726 : Bool;
      HELP_OPERATOR_727 : Bool;
      HELP_OPERATOR_728 : Bool;
      HELP_OPERATOR_729 : Bool;
      HELP_OPERATOR_730 : Bool;
      HELP_OPERATOR_731 : Bool;
      HELP_OPERATOR_732 : Bool;
      HELP_OPERATOR_733 : Bool;
      HELP_OPERATOR_734 : Bool;
      HELP_OPERATOR_735 : Bool;
      HELP_OPERATOR_736 : Bool;
      HELP_OPERATOR_737 : Bool;
      HELP_OPERATOR_738 : Bool;
      HELP_OPERATOR_739 : Bool;
      HELP_OPERATOR_740 : Bool;
      HELP_OPERATOR_741 : Bool;
      HELP_OPERATOR_742 : Bool;
      HELP_OPERATOR_743 : Bool;
      HELP_OPERATOR_744 : Bool;
      HELP_OPERATOR_745 : Bool;
      HELP_OPERATOR_746 : Bool;
      HELP_OPERATOR_747 : Bool;
      HELP_OPERATOR_748 : Bool;
      HELP_OPERATOR_749 : Bool;
      HELP_OPERATOR_750 : Bool;
      HELP_OPERATOR_751 : Bool;
      HELP_OPERATOR_752 : Bool;
      HELP_OPERATOR_753 : Bool;
      HELP_OPERATOR_754 : Bool;
      HELP_OPERATOR_755 : Bool;
      HELP_OPERATOR_756 : Bool;
      HELP_OPERATOR_757 : Bool;
      HELP_OPERATOR_758 : Bool;
      HELP_OPERATOR_759 : Bool;
      HELP_OPERATOR_760 : Bool;
      HELP_OPERATOR_761 : Bool;
      HELP_OPERATOR_762 : Bool;
      HELP_OPERATOR_763 : Bool;
      HELP_OPERATOR_764 : Bool;
      HELP_OPERATOR_765 : Bool;
      HELP_OPERATOR_766 : Bool;
      HELP_OPERATOR_767 : Bool;
      HELP_OPERATOR_768 : Bool;
      HELP_OPERATOR_769 : Bool;
      HELP_OPERATOR_770 : Bool;
      HELP_OPERATOR_771 : Bool;
      HELP_OPERATOR_772 : Bool;
      HELP_OPERATOR_773 : Bool;
      HELP_OPERATOR_774 : Bool;
      HELP_OPERATOR_775 : Bool;
      HELP_OPERATOR_776 : Bool;
      HELP_OPERATOR_777 : Bool;
      HELP_OPERATOR_778 : Bool;
      HELP_OPERATOR_779 : Bool;
      HELP_OPERATOR_780 : Bool;
      HELP_OPERATOR_781 : Bool;
      HELP_OPERATOR_782 : Bool;
      HELP_OPERATOR_783 : Bool;
      HELP_OPERATOR_784 : Bool;
      HELP_OPERATOR_785 : Bool;
      HELP_OPERATOR_786 : Bool;
      HELP_OPERATOR_787 : Bool;
      HELP_OPERATOR_788 : Bool;
      HELP_OPERATOR_789 : Bool;
      HELP_OPERATOR_790 : Bool;
      HELP_OPERATOR_791 : Bool;
      HELP_OPERATOR_792 : Bool;
      HELP_OPERATOR_793 : Bool;
      HELP_OPERATOR_794 : Bool;
      HELP_OPERATOR_795 : Bool;
      HELP_OPERATOR_796 : Bool;
      HELP_OPERATOR_797 : Bool;
      HELP_OPERATOR_798 : Bool;
      HELP_OPERATOR_799 : Bool;
      HELP_OPERATOR_800 : Bool;
      HELP_OPERATOR_801 : Bool;
      HELP_OPERATOR_802 : Bool;
      HELP_OPERATOR_803 : Bool;
      HELP_OPERATOR_804 : Bool;
      HELP_OPERATOR_805 : Bool;
      HELP_OPERATOR_806 : Bool;
      HELP_OPERATOR_807 : Bool;
      HELP_OPERATOR_808 : Bool;
      HELP_OPERATOR_809 : Bool;
      HELP_OPERATOR_810 : Bool;
      HELP_OPERATOR_811 : Bool;
      HELP_OPERATOR_812 : Bool;
      HELP_OPERATOR_813 : Bool;
      HELP_OPERATOR_814 : Bool;
      HELP_OPERATOR_815 : Bool;
      HELP_OPERATOR_816 : Bool;
      HELP_OPERATOR_817 : Bool;
      HELP_OPERATOR_818 : Bool;
      HELP_OPERATOR_819 : Bool;
      HELP_OPERATOR_820 : Bool;
      HELP_OPERATOR_821 : Bool;
      HELP_OPERATOR_822 : Bool;
      HELP_OPERATOR_823 : Bool;
      HELP_OPERATOR_824 : Bool;
      HELP_OPERATOR_825 : Bool;
      HELP_OPERATOR_826 : Bool;
      HELP_OPERATOR_827 : Bool;
      HELP_OPERATOR_828 : Bool;
      HELP_OPERATOR_829 : Bool;
      HELP_OPERATOR_830 : Bool;
      HELP_OPERATOR_831 : Bool;
      HELP_OPERATOR_832 : Bool;
      HELP_OPERATOR_833 : Bool;
      HELP_OPERATOR_834 : Bool;
      HELP_OPERATOR_835 : Bool;
      HELP_OPERATOR_836 : Bool;
      HELP_OPERATOR_837 : Bool;
      HELP_OPERATOR_838 : Bool;
      HELP_OPERATOR_839 : Bool;
      HELP_OPERATOR_840 : Bool;
      HELP_OPERATOR_841 : Bool;
      HELP_OPERATOR_842 : Bool;
      HELP_OPERATOR_843 : Bool;
      HELP_OPERATOR_844 : Bool;
      HELP_OPERATOR_845 : Bool;
      HELP_OPERATOR_846 : Bool;
      HELP_OPERATOR_847 : Bool;
      HELP_OPERATOR_848 : Bool;
      HELP_OPERATOR_849 : Bool;
      HELP_OPERATOR_850 : Bool;
      HELP_OPERATOR_851 : Bool;
      HELP_OPERATOR_852 : Bool;
      HELP_OPERATOR_853 : Bool;
      HELP_OPERATOR_854 : Bool;
      HELP_OPERATOR_855 : Bool;
      HELP_OPERATOR_856 : Bool;
      HELP_OPERATOR_857 : Bool;
      HELP_OPERATOR_858 : Bool;
      HELP_OPERATOR_859 : Bool;
      HELP_OPERATOR_860 : Bool;
      HELP_OPERATOR_861 : Bool;
      HELP_OPERATOR_862 : Bool;
      HELP_OPERATOR_863 : Bool;
      HELP_OPERATOR_864 : Bool;
      HELP_OPERATOR_865 : Bool;
      HELP_OPERATOR_866 : Bool;
      HELP_OPERATOR_867 : Bool;
      HELP_OPERATOR_868 : Bool;
      HELP_OPERATOR_869 : Bool;
      HELP_OPERATOR_870 : Bool;
      HELP_OPERATOR_871 : Bool;
      HELP_OPERATOR_872 : Bool;
      HELP_OPERATOR_873 : Bool;
      HELP_OPERATOR_874 : Bool;
      HELP_OPERATOR_875 : Bool;
      HELP_OPERATOR_876 : Bool;
      HELP_OPERATOR_877 : Bool;
      HELP_OPERATOR_878 : Bool;
      HELP_OPERATOR_879 : Bool;
      HELP_OPERATOR_880 : Bool;
      HELP_OPERATOR_881 : Bool;
      HELP_OPERATOR_882 : Bool;
      HELP_OPERATOR_883 : Bool;
      HELP_OPERATOR_884 : Bool;
      HELP_OPERATOR_885 : Bool;
      HELP_OPERATOR_886 : Bool;
      HELP_OPERATOR_887 : Bool;
      HELP_OPERATOR_888 : Bool;
      HELP_OPERATOR_889 : Bool;
      HELP_OPERATOR_890 : Bool;
      HELP_OPERATOR_891 : Bool;
      HELP_OPERATOR_892 : Bool;
      HELP_OPERATOR_893 : Bool;
      HELP_OPERATOR_894 : Bool;
      HELP_OPERATOR_895 : Bool;
      HELP_OPERATOR_896 : Bool;
      HELP_OPERATOR_897 : Bool;
      HELP_OPERATOR_898 : Bool;
      HELP_OPERATOR_899 : Bool;
      HELP_OPERATOR_900 : Bool;   // RETURN GANTRY TO OUT OF COLLISION POSITION
      HELP_OPERATOR_901 : Bool;   // REQUEST GANTRY TO OPEN SAFETY GATES
      HELP_OPERATOR_902 : Bool;
      HELP_OPERATOR_903 : Bool;
      HELP_OPERATOR_904 : Bool;
      HELP_OPERATOR_905 : Bool;
      HELP_OPERATOR_906 : Bool;
      HELP_OPERATOR_907 : Bool;
      HELP_OPERATOR_908 : Bool;
      HELP_OPERATOR_909 : Bool;
      HELP_OPERATOR_910 : Bool;
      HELP_OPERATOR_911 : Bool;
      HELP_OPERATOR_912 : Bool;
      HELP_OPERATOR_913 : Bool;
      HELP_OPERATOR_914 : Bool;
      HELP_OPERATOR_915 : Bool;
      HELP_OPERATOR_916 : Bool;
      HELP_OPERATOR_917 : Bool;
      HELP_OPERATOR_918 : Bool;
      HELP_OPERATOR_919 : Bool;
      HELP_OPERATOR_920 : Bool;
      HELP_OPERATOR_921 : Bool;
      HELP_OPERATOR_922 : Bool;
      HELP_OPERATOR_923 : Bool;
      HELP_OPERATOR_924 : Bool;
      HELP_OPERATOR_925 : Bool;   // RETURN ROBOT TO OUT OF COLLISION POSITION
      HELP_OPERATOR_926 : Bool;   // REQUEST ROBOT TO OPEN SAFETY GATES
      HELP_OPERATOR_927 : Bool;
      HELP_OPERATOR_928 : Bool;
      HELP_OPERATOR_929 : Bool;
      HELP_OPERATOR_930 : Bool;
      HELP_OPERATOR_931 : Bool;
      HELP_OPERATOR_932 : Bool;
      HELP_OPERATOR_933 : Bool;
      HELP_OPERATOR_934 : Bool;
      HELP_OPERATOR_935 : Bool;
      HELP_OPERATOR_936 : Bool;
      HELP_OPERATOR_937 : Bool;
      HELP_OPERATOR_938 : Bool;
      HELP_OPERATOR_939 : Bool;
      HELP_OPERATOR_940 : Bool;
      HELP_OPERATOR_941 : Bool;
      HELP_OPERATOR_942 : Bool;
      HELP_OPERATOR_943 : Bool;
      HELP_OPERATOR_944 : Bool;
      HELP_OPERATOR_945 : Bool;
      HELP_OPERATOR_946 : Bool;
      HELP_OPERATOR_947 : Bool;
      HELP_OPERATOR_948 : Bool;
      HELP_OPERATOR_949 : Bool;
      HELP_OPERATOR_950 : Bool;
      HELP_OPERATOR_951 : Bool;
      HELP_OPERATOR_952 : Bool;
      HELP_OPERATOR_953 : Bool;
      HELP_OPERATOR_954 : Bool;
      HELP_OPERATOR_955 : Bool;
      HELP_OPERATOR_956 : Bool;
      HELP_OPERATOR_957 : Bool;
      HELP_OPERATOR_958 : Bool;
      HELP_OPERATOR_959 : Bool;
      HELP_OPERATOR_960 : Bool;
      HELP_OPERATOR_961 : Bool;
      HELP_OPERATOR_962 : Bool;
      HELP_OPERATOR_963 : Bool;
      HELP_OPERATOR_964 : Bool;
      HELP_OPERATOR_965 : Bool;
      HELP_OPERATOR_966 : Bool;
      HELP_OPERATOR_967 : Bool;
      HELP_OPERATOR_968 : Bool;
      HELP_OPERATOR_969 : Bool;
      HELP_OPERATOR_970 : Bool;
      HELP_OPERATOR_971 : Bool;
      HELP_OPERATOR_972 : Bool;
      HELP_OPERATOR_973 : Bool;
      HELP_OPERATOR_974 : Bool;
      HELP_OPERATOR_975 : Bool;
      HELP_OPERATOR_976 : Bool;
      HELP_OPERATOR_977 : Bool;
      HELP_OPERATOR_978 : Bool;
      HELP_OPERATOR_979 : Bool;
      HELP_OPERATOR_980 : Bool;
      HELP_OPERATOR_981 : Bool;
      HELP_OPERATOR_982 : Bool;
      HELP_OPERATOR_983 : Bool;
      HELP_OPERATOR_984 : Bool;
      HELP_OPERATOR_985 : Bool;
      HELP_OPERATOR_986 : Bool;
      HELP_OPERATOR_987 : Bool;
      HELP_OPERATOR_988 : Bool;
      HELP_OPERATOR_989 : Bool;
      HELP_OPERATOR_990 : Bool;
      HELP_OPERATOR_991 : Bool;
      HELP_OPERATOR_992 : Bool;
      HELP_OPERATOR_993 : Bool;
      HELP_OPERATOR_994 : Bool;
      HELP_OPERATOR_995 : Bool;
      HELP_OPERATOR_996 : Bool;
      HELP_OPERATOR_997 : Bool;
      HELP_OPERATOR_998 : Bool;
      HELP_OPERATOR_999 : Bool;
      HELP_OPERATOR_1000 : Bool;
   END_VAR
BEGIN
END_DATA_BLOCK
